// TIA Portal V20 export
DATA_BLOCK "InstGetIdentMv"   // DB220
// stored: InstanceOfName GetIdentMv, InstanceOfType FB
"GetIdentMv"
   // VAR_INPUT
   //    identMvAllUnits { ExternalAccessible := 'False'; ExternalVisible := 'False'; ExternalWritable := 'False'} : Array[0.."NO_OF_UNITS"] of "typeEMIdentMv";
   //    numberOfMvReaders : USInt := 1;
   // END_VAR
   // VAR_OUTPUT
   //    selectedUnit : USInt := 1;
   //    selectedEM : USInt := 6;
   //    error : Word := 16#7001;
   // END_VAR
   // VAR_IN_OUT
   //    IdentMvInterfaceHmi : "typeIdentMvHmi";
   // END_VAR
   // VAR
   //    statSelectedEMIdentMv : USInt := 6;
   //    statSelectedUnitIdentRMv : USInt := 1;
   // END_VAR
BEGIN
   identMvAllUnits[0].identMvEM[0..7].selectedUnit := 0;
   identMvAllUnits[0].identMvEM[0..7].selectedEM := 0;
   identMvAllUnits[0].identMvEM[0..7].mvReaderId := 0;
   identMvAllUnits[0].identMvEM[0..7].numberOfMv := 0;
   identMvAllUnits[0].identMvEM[0].mvReader[0..1].deviceName := WSTRING#'';
   identMvAllUnits[0].identMvEM[1].mvReader[0..1].deviceName := WSTRING#'';
   identMvAllUnits[0].identMvEM[2].mvReader[0..1].deviceName := WSTRING#'';
   identMvAllUnits[0].identMvEM[3].mvReader[0..1].deviceName := WSTRING#'';
   identMvAllUnits[0].identMvEM[4].mvReader[0..1].deviceName := WSTRING#'';
   identMvAllUnits[0].identMvEM[5].mvReader[0..1].deviceName := WSTRING#'';
   identMvAllUnits[0].identMvEM[6].mvReader[0..1].deviceName := WSTRING#'';
   identMvAllUnits[0].identMvEM[7].mvReader[0..1].deviceName := WSTRING#'';
   identMvAllUnits[0].identMvEM[0].mvReader[0..1].deviceType := WSTRING#'';
   identMvAllUnits[0].identMvEM[1].mvReader[0..1].deviceType := WSTRING#'';
   identMvAllUnits[0].identMvEM[2].mvReader[0..1].deviceType := WSTRING#'';
   identMvAllUnits[0].identMvEM[3].mvReader[0..1].deviceType := WSTRING#'';
   identMvAllUnits[0].identMvEM[4].mvReader[0..1].deviceType := WSTRING#'';
   identMvAllUnits[0].identMvEM[5].mvReader[0..1].deviceType := WSTRING#'';
   identMvAllUnits[0].identMvEM[6].mvReader[0..1].deviceType := WSTRING#'';
   identMvAllUnits[0].identMvEM[7].mvReader[0..1].deviceType := WSTRING#'';
   identMvAllUnits[0].identMvEM[0].mvReader[0..1].deviceId := 0;
   identMvAllUnits[0].identMvEM[1].mvReader[0..1].deviceId := 0;
   identMvAllUnits[0].identMvEM[2].mvReader[0..1].deviceId := 0;
   identMvAllUnits[0].identMvEM[3].mvReader[0..1].deviceId := 0;
   identMvAllUnits[0].identMvEM[4].mvReader[0..1].deviceId := 0;
   identMvAllUnits[0].identMvEM[5].mvReader[0..1].deviceId := 0;
   identMvAllUnits[0].identMvEM[6].mvReader[0..1].deviceId := 0;
   identMvAllUnits[0].identMvEM[7].mvReader[0..1].deviceId := 0;
   identMvAllUnits[0].identMvEM[0].mvReader[0..1].tagType := WSTRING#'';
   identMvAllUnits[0].identMvEM[1].mvReader[0..1].tagType := WSTRING#'';
   identMvAllUnits[0].identMvEM[2].mvReader[0..1].tagType := WSTRING#'';
   identMvAllUnits[0].identMvEM[3].mvReader[0..1].tagType := WSTRING#'';
   identMvAllUnits[0].identMvEM[4].mvReader[0..1].tagType := WSTRING#'';
   identMvAllUnits[0].identMvEM[5].mvReader[0..1].tagType := WSTRING#'';
   identMvAllUnits[0].identMvEM[6].mvReader[0..1].tagType := WSTRING#'';
   identMvAllUnits[0].identMvEM[7].mvReader[0..1].tagType := WSTRING#'';
   identMvAllUnits[0].identMvEM[0].mvReader[0..1].cameraMode := WSTRING#'';
   identMvAllUnits[0].identMvEM[1].mvReader[0..1].cameraMode := WSTRING#'';
   identMvAllUnits[0].identMvEM[2].mvReader[0..1].cameraMode := WSTRING#'';
   identMvAllUnits[0].identMvEM[3].mvReader[0..1].cameraMode := WSTRING#'';
   identMvAllUnits[0].identMvEM[4].mvReader[0..1].cameraMode := WSTRING#'';
   identMvAllUnits[0].identMvEM[5].mvReader[0..1].cameraMode := WSTRING#'';
   identMvAllUnits[0].identMvEM[6].mvReader[0..1].cameraMode := WSTRING#'';
   identMvAllUnits[0].identMvEM[7].mvReader[0..1].cameraMode := WSTRING#'';
   identMvAllUnits[0].identMvEM[0].mvReader[0..1].resultState := WSTRING#'';
   identMvAllUnits[0].identMvEM[1].mvReader[0..1].resultState := WSTRING#'';
   identMvAllUnits[0].identMvEM[2].mvReader[0..1].resultState := WSTRING#'';
   identMvAllUnits[0].identMvEM[3].mvReader[0..1].resultState := WSTRING#'';
   identMvAllUnits[0].identMvEM[4].mvReader[0..1].resultState := WSTRING#'';
   identMvAllUnits[0].identMvEM[5].mvReader[0..1].resultState := WSTRING#'';
   identMvAllUnits[0].identMvEM[6].mvReader[0..1].resultState := WSTRING#'';
   identMvAllUnits[0].identMvEM[7].mvReader[0..1].resultState := WSTRING#'';
   identMvAllUnits[0].identMvEM[0].mvReader[0..1].progNo := 0;
   identMvAllUnits[0].identMvEM[1].mvReader[0..1].progNo := 0;
   identMvAllUnits[0].identMvEM[2].mvReader[0..1].progNo := 0;
   identMvAllUnits[0].identMvEM[3].mvReader[0..1].progNo := 0;
   identMvAllUnits[0].identMvEM[4].mvReader[0..1].progNo := 0;
   identMvAllUnits[0].identMvEM[5].mvReader[0..1].progNo := 0;
   identMvAllUnits[0].identMvEM[6].mvReader[0..1].progNo := 0;
   identMvAllUnits[0].identMvEM[7].mvReader[0..1].progNo := 0;
   identMvAllUnits[0].identMvEM[0].mvReader[0..1].progNumberWrite := 0;
   identMvAllUnits[0].identMvEM[1].mvReader[0..1].progNumberWrite := 0;
   identMvAllUnits[0].identMvEM[2].mvReader[0..1].progNumberWrite := 0;
   identMvAllUnits[0].identMvEM[3].mvReader[0..1].progNumberWrite := 0;
   identMvAllUnits[0].identMvEM[4].mvReader[0..1].progNumberWrite := 0;
   identMvAllUnits[0].identMvEM[5].mvReader[0..1].progNumberWrite := 0;
   identMvAllUnits[0].identMvEM[6].mvReader[0..1].progNumberWrite := 0;
   identMvAllUnits[0].identMvEM[7].mvReader[0..1].progNumberWrite := 0;
   identMvAllUnits[0].identMvEM[0].mvReader[0..1].pushbutton := 16#0000;
   identMvAllUnits[0].identMvEM[1].mvReader[0..1].pushbutton := 16#0000;
   identMvAllUnits[0].identMvEM[2].mvReader[0..1].pushbutton := 16#0000;
   identMvAllUnits[0].identMvEM[3].mvReader[0..1].pushbutton := 16#0000;
   identMvAllUnits[0].identMvEM[4].mvReader[0..1].pushbutton := 16#0000;
   identMvAllUnits[0].identMvEM[5].mvReader[0..1].pushbutton := 16#0000;
   identMvAllUnits[0].identMvEM[6].mvReader[0..1].pushbutton := 16#0000;
   identMvAllUnits[0].identMvEM[7].mvReader[0..1].pushbutton := 16#0000;
   identMvAllUnits[0].identMvEM[0].mvReader[0..1].enablePushbutton := 16#0000;
   identMvAllUnits[0].identMvEM[1].mvReader[0..1].enablePushbutton := 16#0000;
   identMvAllUnits[0].identMvEM[2].mvReader[0..1].enablePushbutton := 16#0000;
   identMvAllUnits[0].identMvEM[3].mvReader[0..1].enablePushbutton := 16#0000;
   identMvAllUnits[0].identMvEM[4].mvReader[0..1].enablePushbutton := 16#0000;
   identMvAllUnits[0].identMvEM[5].mvReader[0..1].enablePushbutton := 16#0000;
   identMvAllUnits[0].identMvEM[6].mvReader[0..1].enablePushbutton := 16#0000;
   identMvAllUnits[0].identMvEM[7].mvReader[0..1].enablePushbutton := 16#0000;
   identMvAllUnits[0].identMvEM[0].mvReader[0..1].status := 16#0000;
   identMvAllUnits[0].identMvEM[1].mvReader[0..1].status := 16#0000;
   identMvAllUnits[0].identMvEM[2].mvReader[0..1].status := 16#0000;
   identMvAllUnits[0].identMvEM[3].mvReader[0..1].status := 16#0000;
   identMvAllUnits[0].identMvEM[4].mvReader[0..1].status := 16#0000;
   identMvAllUnits[0].identMvEM[5].mvReader[0..1].status := 16#0000;
   identMvAllUnits[0].identMvEM[6].mvReader[0..1].status := 16#0000;
   identMvAllUnits[0].identMvEM[7].mvReader[0..1].status := 16#0000;
   identMvAllUnits[0].identMvEM[0].mvReader[0..1].alarmCategorie := 0;
   identMvAllUnits[0].identMvEM[1].mvReader[0..1].alarmCategorie := 0;
   identMvAllUnits[0].identMvEM[2].mvReader[0..1].alarmCategorie := 0;
   identMvAllUnits[0].identMvEM[3].mvReader[0..1].alarmCategorie := 0;
   identMvAllUnits[0].identMvEM[4].mvReader[0..1].alarmCategorie := 0;
   identMvAllUnits[0].identMvEM[5].mvReader[0..1].alarmCategorie := 0;
   identMvAllUnits[0].identMvEM[6].mvReader[0..1].alarmCategorie := 0;
   identMvAllUnits[0].identMvEM[7].mvReader[0..1].alarmCategorie := 0;
   identMvAllUnits[0].identMvEM[0].mvReader[0..1].alarmNo := 0;
   identMvAllUnits[0].identMvEM[1].mvReader[0..1].alarmNo := 0;
   identMvAllUnits[0].identMvEM[2].mvReader[0..1].alarmNo := 0;
   identMvAllUnits[0].identMvEM[3].mvReader[0..1].alarmNo := 0;
   identMvAllUnits[0].identMvEM[4].mvReader[0..1].alarmNo := 0;
   identMvAllUnits[0].identMvEM[5].mvReader[0..1].alarmNo := 0;
   identMvAllUnits[0].identMvEM[6].mvReader[0..1].alarmNo := 0;
   identMvAllUnits[0].identMvEM[7].mvReader[0..1].alarmNo := 0;
   identMvAllUnits[0].identMvEM[0].mvReader[0..1].alarmCode := 16#0000_0000;
   identMvAllUnits[0].identMvEM[1].mvReader[0..1].alarmCode := 16#0000_0000;
   identMvAllUnits[0].identMvEM[2].mvReader[0..1].alarmCode := 16#0000_0000;
   identMvAllUnits[0].identMvEM[3].mvReader[0..1].alarmCode := 16#0000_0000;
   identMvAllUnits[0].identMvEM[4].mvReader[0..1].alarmCode := 16#0000_0000;
   identMvAllUnits[0].identMvEM[5].mvReader[0..1].alarmCode := 16#0000_0000;
   identMvAllUnits[0].identMvEM[6].mvReader[0..1].alarmCode := 16#0000_0000;
   identMvAllUnits[0].identMvEM[7].mvReader[0..1].alarmCode := 16#0000_0000;
   identMvAllUnits[0].identMvEM[0].mvReader[0..1].resultColor := 0;
   identMvAllUnits[0].identMvEM[1].mvReader[0..1].resultColor := 0;
   identMvAllUnits[0].identMvEM[2].mvReader[0..1].resultColor := 0;
   identMvAllUnits[0].identMvEM[3].mvReader[0..1].resultColor := 0;
   identMvAllUnits[0].identMvEM[4].mvReader[0..1].resultColor := 0;
   identMvAllUnits[0].identMvEM[5].mvReader[0..1].resultColor := 0;
   identMvAllUnits[0].identMvEM[6].mvReader[0..1].resultColor := 0;
   identMvAllUnits[0].identMvEM[7].mvReader[0..1].resultColor := 0;
   identMvAllUnits[0].identMvEM[0].mvReader[0..1].statusColorCode := 0;
   identMvAllUnits[0].identMvEM[1].mvReader[0..1].statusColorCode := 0;
   identMvAllUnits[0].identMvEM[2].mvReader[0..1].statusColorCode := 0;
   identMvAllUnits[0].identMvEM[3].mvReader[0..1].statusColorCode := 0;
   identMvAllUnits[0].identMvEM[4].mvReader[0..1].statusColorCode := 0;
   identMvAllUnits[0].identMvEM[5].mvReader[0..1].statusColorCode := 0;
   identMvAllUnits[0].identMvEM[6].mvReader[0..1].statusColorCode := 0;
   identMvAllUnits[0].identMvEM[7].mvReader[0..1].statusColorCode := 0;
   identMvAllUnits[0].identMvEM[0].mvReader[0..1].datRead1 := '';
   identMvAllUnits[0].identMvEM[1].mvReader[0..1].datRead1 := '';
   identMvAllUnits[0].identMvEM[2].mvReader[0..1].datRead1 := '';
   identMvAllUnits[0].identMvEM[3].mvReader[0..1].datRead1 := '';
   identMvAllUnits[0].identMvEM[4].mvReader[0..1].datRead1 := '';
   identMvAllUnits[0].identMvEM[5].mvReader[0..1].datRead1 := '';
   identMvAllUnits[0].identMvEM[6].mvReader[0..1].datRead1 := '';
   identMvAllUnits[0].identMvEM[7].mvReader[0..1].datRead1 := '';
   identMvAllUnits[0].identMvEM[0].mvReader[0..1].datRead2 := '';
   identMvAllUnits[0].identMvEM[1].mvReader[0..1].datRead2 := '';
   identMvAllUnits[0].identMvEM[2].mvReader[0..1].datRead2 := '';
   identMvAllUnits[0].identMvEM[3].mvReader[0..1].datRead2 := '';
   identMvAllUnits[0].identMvEM[4].mvReader[0..1].datRead2 := '';
   identMvAllUnits[0].identMvEM[5].mvReader[0..1].datRead2 := '';
   identMvAllUnits[0].identMvEM[6].mvReader[0..1].datRead2 := '';
   identMvAllUnits[0].identMvEM[7].mvReader[0..1].datRead2 := '';
   identMvAllUnits[0].identMvEM[0].mvReader[0..1].datRead3 := '';
   identMvAllUnits[0].identMvEM[1].mvReader[0..1].datRead3 := '';
   identMvAllUnits[0].identMvEM[2].mvReader[0..1].datRead3 := '';
   identMvAllUnits[0].identMvEM[3].mvReader[0..1].datRead3 := '';
   identMvAllUnits[0].identMvEM[4].mvReader[0..1].datRead3 := '';
   identMvAllUnits[0].identMvEM[5].mvReader[0..1].datRead3 := '';
   identMvAllUnits[0].identMvEM[6].mvReader[0..1].datRead3 := '';
   identMvAllUnits[0].identMvEM[7].mvReader[0..1].datRead3 := '';
   identMvAllUnits[0].identMvEM[0].mvReader[0..1].datRead4 := '';
   identMvAllUnits[0].identMvEM[1].mvReader[0..1].datRead4 := '';
   identMvAllUnits[0].identMvEM[2].mvReader[0..1].datRead4 := '';
   identMvAllUnits[0].identMvEM[3].mvReader[0..1].datRead4 := '';
   identMvAllUnits[0].identMvEM[4].mvReader[0..1].datRead4 := '';
   identMvAllUnits[0].identMvEM[5].mvReader[0..1].datRead4 := '';
   identMvAllUnits[0].identMvEM[6].mvReader[0..1].datRead4 := '';
   identMvAllUnits[0].identMvEM[7].mvReader[0..1].datRead4 := '';
   identMvAllUnits[0].identMvEM[0].mvReader[0].datWrite1 := '';
   identMvAllUnits[0].identMvEM[0].mvReader[1].datWrite1 := 'Siemens';
   identMvAllUnits[0].identMvEM[1].mvReader[0..1].datWrite1 := '';
   identMvAllUnits[0].identMvEM[2].mvReader[0..1].datWrite1 := '';
   identMvAllUnits[0].identMvEM[3].mvReader[0..1].datWrite1 := '';
   identMvAllUnits[0].identMvEM[4].mvReader[0..1].datWrite1 := '';
   identMvAllUnits[0].identMvEM[5].mvReader[0..1].datWrite1 := '';
   identMvAllUnits[0].identMvEM[6].mvReader[0..1].datWrite1 := '';
   identMvAllUnits[0].identMvEM[7].mvReader[0..1].datWrite1 := '';
   identMvAllUnits[0].identMvEM[0].mvReader[0..1].datWrite2 := '';
   identMvAllUnits[0].identMvEM[1].mvReader[0..1].datWrite2 := '';
   identMvAllUnits[0].identMvEM[2].mvReader[0..1].datWrite2 := '';
   identMvAllUnits[0].identMvEM[3].mvReader[0..1].datWrite2 := '';
   identMvAllUnits[0].identMvEM[4].mvReader[0..1].datWrite2 := '';
   identMvAllUnits[0].identMvEM[5].mvReader[0..1].datWrite2 := '';
   identMvAllUnits[0].identMvEM[6].mvReader[0..1].datWrite2 := '';
   identMvAllUnits[0].identMvEM[7].mvReader[0..1].datWrite2 := '';
   identMvAllUnits[0].identMvEM[0].mvReader[0..1].datWrite3 := '';
   identMvAllUnits[0].identMvEM[1].mvReader[0..1].datWrite3 := '';
   identMvAllUnits[0].identMvEM[2].mvReader[0..1].datWrite3 := '';
   identMvAllUnits[0].identMvEM[3].mvReader[0..1].datWrite3 := '';
   identMvAllUnits[0].identMvEM[4].mvReader[0..1].datWrite3 := '';
   identMvAllUnits[0].identMvEM[5].mvReader[0..1].datWrite3 := '';
   identMvAllUnits[0].identMvEM[6].mvReader[0..1].datWrite3 := '';
   identMvAllUnits[0].identMvEM[7].mvReader[0..1].datWrite3 := '';
   identMvAllUnits[0].identMvEM[0].mvReader[0..1].datWrite4 := '';
   identMvAllUnits[0].identMvEM[1].mvReader[0..1].datWrite4 := '';
   identMvAllUnits[0].identMvEM[2].mvReader[0..1].datWrite4 := '';
   identMvAllUnits[0].identMvEM[3].mvReader[0..1].datWrite4 := '';
   identMvAllUnits[0].identMvEM[4].mvReader[0..1].datWrite4 := '';
   identMvAllUnits[0].identMvEM[5].mvReader[0..1].datWrite4 := '';
   identMvAllUnits[0].identMvEM[6].mvReader[0..1].datWrite4 := '';
   identMvAllUnits[0].identMvEM[7].mvReader[0..1].datWrite4 := '';
END_DATA_BLOCK
